SUBAPPLICATION SystemTickSender_ISO_OPC (* SystemTick-Heartbeat auf VT-Zahlenfeld anzeigen UND per OPC-UA publizieren *)
  (* Standard: 61499-2; Description: Copyright (c) 2026 Meisterschulen am Ostbahnhof This program and the accompanying materials are made available under the terms of the Eclipse Public License 2.0 which is available at https://www.eclipse.org/legal/epl-2.0/ SPDX-License-Identifier: EPL-2.0 *)
  (* Version 1.0, 2026-08-07, Franz Höpfinger, Meisterschulen am Ostbahnhof, initial API and implementation and/or initial documentation *)
  PACKAGE MyLib::sys;
  IMPORT isobus::UT::Q::const::IDs::ID_NULL;
  (* Documentation:
  SystemTick-Heartbeat lokal auf VT anzeigen UND per OPC-UA publizieren
   Kombiniert SystemTickSender_ISO (Anzeige auf einem lokalen VT-Zahlenfeld) mit SystemTickSender_OPC (Remote-Publish per OPC-UA), damit dasselbe Lebenszeichen sowohl am eigenen Bildschirm sichtbar ist als auch von anderen Modulen per Remote-Subscribe überwacht werden kann.
   Funktionsbeschreibung
    - System_Tick liefert den Zählerstand als ADI.
   - ADI_SPLIT_2 verteilt dieses eine Signal auf zwei Ziele, weil ein Adapter-Socket nur eine Quelle annehmen kann.
   - ADI_TO_AUDI → Q_NumericValue_AUDI (u16ObjId) zeigt den Wert lokal auf dem VT an - wie bei SystemTickSender_ISO.
   - ADI_PUBLISH_1 (ID_WRITE) veröffentlicht denselben Wert per OPC-UA - wie bei SystemTickSender_OPC.
    Wird nur eine der beiden Ausgaben gebraucht, die einfachere SystemTickSender_ISO (nur VT) bzw. SystemTickSender_OPC (nur OPC-UA) verwenden.
  *)
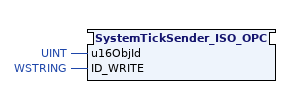
  VAR_INPUT
    u16ObjId : UINT := ID_NULL; (* Object ID VT-Zahlenausgabefeld (OutputNumberField), zeigt den Tick-Zaehlerstand an *)
    ID_WRITE : WSTRING; (* OPC-UA Publish-Key fuer den Tick-Zaehlerstand (fuer Remote-Subscribe durch andere Module) *)
  END_VAR
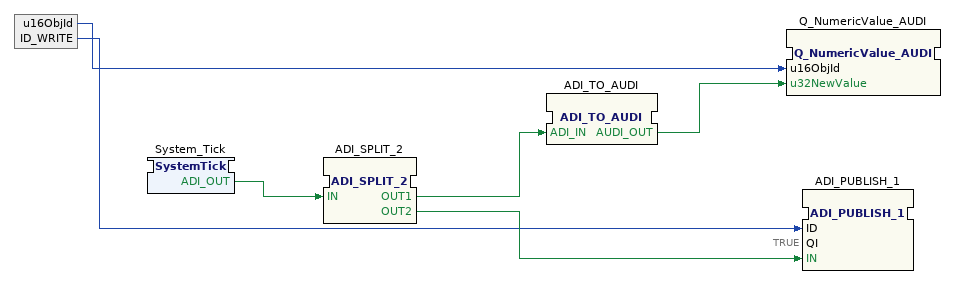
  FBS
    Q_NumericValue_AUDI : isobus::UT::Q::Q_NumericValue_AUDI;
    ADI_SPLIT_2 : adapter::events::unidirectional::ADI_SPLIT_2;
    ADI_TO_AUDI : adapter::conversion::unidirectional::ADI_TO_AUDI;
    ADI_PUBLISH_1 : adapter::net::ADI_PUBLISH_1(QI := TRUE);
  END_FBS
  SUBAPPS
    System_Tick : MyLib::sys::SystemTick;
  END_SUBAPPS
  DATA_CONNECTIONS
    u16ObjId TO Q_NumericValue_AUDI.u16ObjId;
    ID_WRITE TO ADI_PUBLISH_1.ID;
  END_CONNECTIONS
  ADAPTER_CONNECTIONS
    System_Tick.ADI_OUT TO ADI_SPLIT_2.IN;
    ADI_TO_AUDI.AUDI_OUT TO Q_NumericValue_AUDI.u32NewValue;
    ADI_SPLIT_2.OUT1 TO ADI_TO_AUDI.ADI_IN;
    ADI_SPLIT_2.OUT2 TO ADI_PUBLISH_1.IN;
  END_CONNECTIONS
END_SUBAPPLICATION
